RoboDK station: Ruta_IZQ.rdk

Station Ruta_IZQ (saved by RoboDK 5.5.4). Poses are relative to the parent item; angles as X-Y-Z fixed-axis rotations.
  - object Ruta_IZQ at (0, 0, 0) mm, geometry from Curva importada
